Staubli VAL3: listins.pgx

public program listins(string& x_sItems[] (dimensions=1), num x_nPos (dimensions=1))
  local num i
  local num l_nSize
begin
  //
  // Staubli Copyright 2005
  //
  l_nSize=size(sItems)-1
  if ((x_nPos>=0) and (x_nPos<=l_nSize))
    for i=0 to (size(x_sItems)-1)
      if size(sItems)!=1 or sItems!=""
        insert(sItems[x_nPos+i])
        insert(bReadWrite[x_nPos+i])
      endIf
      sItems[x_nPos+i]=x_sItems[i]
      // for default the RW is true
      bReadWrite[x_nPos+i]=true
    endFor
  else
    call listadd(x_sItems)
  endIf
end
